// TIA Portal V19 export
DATA_BLOCK "CallEquipment_DB"   // DB151
{ DB_Accessible_From_OPC_UA := 'FALSE' }
// stored: AssignedProDiagFB Unit.Em0.ProDiag, DBAccessibleFromOPCUA false, DBAccessibleFromWebserver false, InstanceOfName Unit.Em0.CallEquipment, InstanceOfType FB, Namespace Unit.Em0
"Unit.Em0.CallEquipment"
   // VAR_IN_OUT
   //    unitStatus : "LAF_typeUnitStatus";
   //    emFeedback : "LUC_typeEmFeedback";
   //    unitAlarmDB : "LAF_typeAlarms";
   // END_VAR
   // VAR
   //    statUnitStatus { ExternalWritable := 'False'} : "LAF_typeUnitStatus";
   //    instManageAlarms { ExternalWritable := 'False'} : "LAF_ManageAlarms";
   // END_VAR
BEGIN
END_DATA_BLOCK
